TYPE ST_JointAxis :
STRUCT
	stAbsEncoderAxisRef	: AXIS_REF;
	stIncEncoderAxisRef	: AXIS_REF;
	bForceSetup : BOOL;
	
	//Bools to determine the type of joint
	bDualEncoderJoint : BOOL;
	bVariableOffsetJoint : BOOL;
	bSingleIncrementalJoint : BOOL;
	bSingleAbsoluteJoint : BOOL;

	
END_STRUCT
END_TYPE

(* stored: Version 1.1.0.1, ProductVersion 3.1.4024.12
   DUT ST_JointAxis: Id {aadcc87d-cf4a-45d7-8196-3b236aafd473} *)
